PROGRAM MAIN
VAR	
	onTimer : TON;
	OffTimer :TOF;
	timerStart : BOOL;
	reverseSignal : BOOL;
	bWatch : BOOL;
	
	onTimer_tune  : TON;
	OffTimer_tune :TOF;
	reverseSignal_tune : BOOL;
END_VAR


(* watch dogs : 10s 간격으로 on/ off *)

onTimer(IN := OffTimer.Q, PT := T#10S);
IF onTimer.Q THEN
  reverseSignal := FALSE;
  mgbl.master_bWatch := FALSE;
ELSE
  reverseSignal := TRUE;
  mgbl.master_bWatch := TRUE;
END_IF
OffTimer(IN := reverseSignal, PT := T#10S);



(* 
mgbl.master_tuning_mode = tune set
tune set :  true -> master, slave호출
tune set :  false -> slave만 호출
*)

master();

slave();

(*
 아래 코드는 Tune Mode Start 후 바로 False로 변경되어 Master 호출이 안됩니다.
 튜닝 완료 후 FALSE로 변경하세요
*)

(*
IF mgbl.master_tuning_mode THEN
	master();
	slave();
	
  (* 튜닝 시간 설정 = mgbl.master_tuning_time *)
    onTimer_tune(IN := OffTimer_tune.Q, PT := LREAL_TO_TIME(mgbl.master_tuning_time)*60000);
    IF onTimer_tune.Q THEN
	  mgbl.master_tuning_mode := FALSE;
	  reverseSignal_tune := FALSE;
	ELSE
	  reverseSignal_tune := TRUE;
    END_IF
    OffTimer_tune(IN := reverseSignal_tune, PT := LREAL_TO_TIME(mgbl.master_tuning_time)*60000);
ELSE
	slave();
END_IF
*)

END_PROGRAM

(* stored: Version 1.1.0.1, ProductVersion 3.1.4024.4
   POU MAIN: Id {c7996b60-7a70-413b-abcb-6b6ff75a050d}, SpecialFunc None *)
